// LS Electric XG5000 project: 67_1
// PLC NewPLC
// module base 0 slot 0: 입출력 모듈:XBC-DN/DP14E (DC 24V 입력 8점, 트랜지스터 출력 6점)

PROGRAM NewProgram (task: 스캔 프로그램)

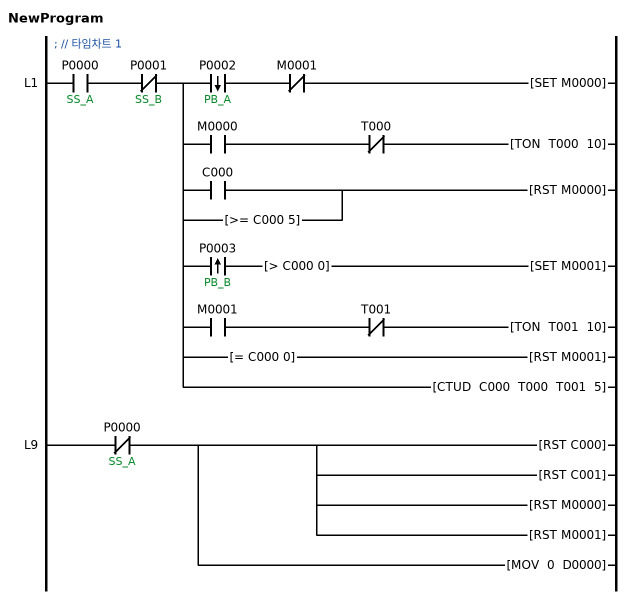
// // 타임차트 1
; L1
LOAD      P0000	// SS_A
AND NOT   P0001	// SS_B
MPUSH
ANDN      P0002	// PB_A
AND NOT   M0001
SET       M0000
MLOAD
AND       M0000
AND NOT   T000
TON       T000 10
MLOAD
LOAD      C000
OR>=      C000 5
AND LOAD
RST       M0000
MLOAD
ANDP      P0003	// PB_B
AND>      C000 0
SET       M0001
MLOAD
AND       M0001
AND NOT   T001
TON       T001 10
MLOAD
AND=      C000 0
RST       M0001
MPOP
CTUD      C000 T000 T001 5
; L9
LOAD NOT  P0000	// SS_A
RST       C000
RST       C001
RST       M0000
RST       M0001
MOV       0 D0000

VARIABLES AND COMMENTS (devices not used above)
P00004	BIT	PB_C
P00040	BIT	PL_A
P00041	BIT	PL_B
P00042	BIT	PL_C
P00043	BIT	PL_D
P00044	BIT	PL_E